FUNCTION_BLOCK FB_CsvlPersistentEventStorage IMPLEMENTS I_PersistentEventStorage
VAR
	fbFileOpen : FB_FileOpen := (sPathName := 'C:\Events.log', nMode := FOPEN_MODEAPPEND OR FOPEN_MODETEXT);
	fbFilePuts : FB_FilePuts;
	fbFileClose : FB_FileClose;
	eWriteState : (FILE_OPEN_TRIGGER ,FILE_OPEN, WAIT_FOR_EVENT, WRITE_EVENT_TRIGGER, WRITE_EVENT, CLOSE_FILE_TRIGGER, CLOSE_FILE, Error);
	stEventWrittenToFile : ST_Event;
	
	CsvString : T_MaxString;
END_VAR

CASE eWriteState OF
	FILE_OPEN_TRIGGER:
		fbFileOpen(bExecute := TRUE);
		eWriteState := FILE_OPEN;
	
	FILE_OPEN:
		fbFileOpen(bExecute := FALSE);
		IF fbFileOpen.bError THEN
			eWriteState := Error;
		ELSIF NOT fbFileOpen.bBusy AND fbFileOpen.hFile <> 0 THEN
			eWriteState := WAIT_FOR_EVENT;
		END_IF
	
	WAIT_FOR_EVENT:
		//
	WRITE_EVENT_TRIGGER:
		CsvString := CreateCsvString(stEvent := stEventWrittenToFile);
		fbFilePuts(bExecute := TRUE, sLine := CsvString, hFile := fbFileOpen.hFile);
		eWriteState := WRITE_EVENT;
	WRITE_EVENT:
		fbFilePuts(bExecute := FALSE);
		IF fbFilePuts.bError THEN
			eWriteState := Error;
		ELSIF NOT fbFileOpen.bBusy THEN
			eWriteState := CLOSE_FILE_TRIGGER;
		END_IF
	CLOSE_FILE_TRIGGER:
		fbFileClose(bExecute := TRUE, hFile := fbFileOpen.hFile);
		eWriteState := CLOSE_FILE;
	CLOSE_FILE:
		fbFileClose(bExecute := FALSE);
		IF fbFileClose.bError THEN
			eWriteState := Error;
		ELSIF NOT fbFileClose.bBusy THEN
			eWriteState := FILE_OPEN_TRIGGER;
		END_IF
	Error:
	//
	
END_CASE

METHOD PRIVATE CreateCsvString : T_MaxString
VAR_INPUT
	stEvent : REFERENCE TO ST_Event;
END_VAR
VAR
	tempString : T_MaxString;
END_VAR
tempString := TO_STRING(stEvent.eEventType);
tempString := CONCAT(STR1:= tempString, STR2:= ',');
tempString := CONCAT(STR1:= tempString, STR2:= TO_STRING(stEvent.eEventSeverity));
tempString := CONCAT(STR1:= tempString, STR2:= ',');
tempString := CONCAT(STR1:= tempString, STR2:= TO_STRING(stEvent.nEventIdentity));
tempString := CONCAT(STR1:= tempString, STR2:= ',');
tempString := CONCAT(STR1:= tempString, STR2:= stEvent.sEventText);
tempString := CONCAT(STR1:= tempString, STR2:= ',');
tempString := CONCAT(STR1:= tempString, STR2:= TO_STRING(stEvent.dtTimeStamp));
tempString := CONCAT(STR1:= tempString, STR2:= '$n'); // special charecter for next line

CreateCsvString := tempString; // output of method equals its name
END_METHOD

METHOD StoreEvent // error: because Interface just describes the behavior nothing about implementation
VAR_INPUT
	stEvent	: ST_Event;
END_VAR
IF eWriteState = WAIT_FOR_EVENT THEN
	eWriteState := WRITE_EVENT_TRIGGER;
	stEventWrittenToFile := stEvent;
END_IF
END_METHOD

END_FUNCTION_BLOCK

(* stored: Version 1.1.0.1, ProductVersion 3.1.4024.12
   POU FB_CsvlPersistentEventStorage: Id {e3547434-c820-42dd-b441-b47298ea1dbf}, SpecialFunc None
   Method CreateCsvString: Id {31115463-8099-412b-893a-d20a6c8301e3}
   Method StoreEvent: Id {51a4c073-b24d-4018-b148-ff0fcf2f7fba} *)
